// TwinCAT 3 PLC project PLC1
// ProgramVersion: 3.1.4024.0
// libraries:
//   Tc2_Standard, * (Beckhoff Automation GmbH)
//   Tc2_System, * (Beckhoff Automation GmbH)
//   Tc3_Module, * (Beckhoff Automation GmbH)
// project tree:
//   CSL/Enums/ E_Step.TcTLEO
//   CSL/FB/ FB_MSF_Pistons.TcPOU
//   CSL/Structs/ ST_CSL_RawOut.TcDUT, ST_CSL_In.TcDUT, ST_CSL_Out.TcDUT, ST_CSL_Params.TcDUT, ST_CSL_RawIn.TcDUT
//   / PlcTask.TcTTO
//   POUs/ MAIN.TcPOU
// real-time tasks:
//   TASK PlcTask: cycle T#10ms, priority 20, ADS port 350
// motion (NC):
//   TASK NC-Task 1 SAF: cycle T#2ms, priority 4, ADS port 501
//   TASK NC-Task 1 SVB: cycle T#10ms, priority 8, ADS port 511
//   AXIS Asse 1 (id 1)
//     OtherSettings: AllowMotionCmdToSlave=true
//     encoder EncType=4
//       EncPara: MaxCount=#x0000ffff
//         Inc: RefSoftSyncMask=#x0000ffff
//     drive DrvType=24
//       Analog: TorqueSetpointScale=10, ScaleFactorActTorque=0.1
//       TimeComp: TaskDelayCycles=1
//     controller CtrType=1
//       CtrPara: PriorControlFactor=1
//         Observer: BandWidth=20
//   AXIS Asse 2 (id 2)
//     OtherSettings: AllowMotionCmdToSlave=true
//     encoder EncType=4
//       EncPara: MaxCount=#x0000ffff
//         Inc: RefSoftSyncMask=#x0000ffff
//     drive DrvType=24
//       Analog: TorqueSetpointScale=10, ScaleFactorActTorque=0.1
//       TimeComp: TaskDelayCycles=1
//     controller CtrType=1
//       CtrPara: PriorControlFactor=1
//         Observer: BandWidth=20
//   AXIS Asse 3 (id 3)
//     OtherSettings: AllowMotionCmdToSlave=true
//     encoder EncType=4
//       EncPara: MaxCount=#x0000ffff
//         Inc: RefSoftSyncMask=#x0000ffff
//     drive DrvType=24
//       Analog: TorqueSetpointScale=10, ScaleFactorActTorque=0.1
//       TimeComp: TaskDelayCycles=1
//     controller CtrType=1
//       CtrPara: PriorControlFactor=1
//         Observer: BandWidth=20
// I/O:
//   DEVICE Dispositivo 1 (EtherCAT), AmsNetId 5.85.197.242.2.1
//     Terminale 1 (EK1200) [EK1200-5000 EtherCAT Power supply (2A E-Bus)]
//       Terminale 2 (EL1809) [EL1809 16Ch. Dig. Input 24V, 3ms]
//       Terminale 3 (EL2809) [EL2809 16Ch. Dig. Output 24V, 0.5A]
//       Terminale 4 (EL3201) [EL3201 1Ch. Ana. Input PT100 (RTD)]
//       Terminale 5 (EL3311) [EL3311 1Ch. Ana. Input Thermocouple (TC)]
//       Terminale 6 (EL3004) [EL3004 4Ch. Ana. Input +/-10V]
//       Terminale 7 (EL1918) [EL1918, 8Ch. Safety Input 24V, TwinSAFE]
//         modules: Module 1 (FSOE), Module 2 (FSLOGIC)
//       Terminale 8 (EL2904) [EL2904, 4 Ch. Safety Output 24V, 0.5A, TwinSAFE]
//         modules: Module 1 (FSOES), Module 2 (DO)
//       Terminale 9 (EL9011) [EL9011 End Terminal]
//   DEVICE Dispositivo 4 (EtherCAT), AmsNetId 5.85.197.242.5.1
//     Terminale 10 (EK1100) [EK1100 EtherCAT Coupler (2A E-Bus)]
//       Terminale 11 (EL1809) [EL1809 16Ch. Dig. Input 24V, 3ms]
//       Terminale 12 (EL2809) [EL2809 16Ch. Dig. Output 24V, 0.5A]
//       Terminale 13 (EL1809) [EL1809 16Ch. Dig. Input 24V, 3ms]
//       Terminale 14 (EL2809-0015) [EL2809-0015 16Ch. Dig. Output 24V DC, 0.35A, not short-circuit proof]
//       Terminale 15 (EL3202) [EL3202 2Ch. Ana. Input PT100 (RTD)]
//       Terminale 16 (EL3312) [EL3312 2Ch. Ana. Input Thermocouple (TC)]
//       Terminale 17 (EL3632) [EL3632 2Ch. IEPE Sensor]
//       Terminale 18 (EL7031) [EL7031 1Ch. Stepper motor output stage (24V, 1.5A)]
//       Terminale 10 (EL9011) [EL9011 End Terminal]
// variable links:
//   NC-Task 1 SAF/Axes/Asse 3 <-> Device 4 (EtherCAT)/Term 10 (EK1100)/Term 18 (EL7031)
//     Drive/Inputs/In/nState1 @bit 3 <-> STM Status/Status/Error
//     Drive/Inputs/In/nState1 @bit 5 <-> STM Status/Status/Moving negative
//     Drive/Inputs/In/nState1 @bit 4 <-> STM Status/Status/Moving positive
//     Drive/Inputs/In/nState1 @bit 1 <-> STM Status/Status/Ready
//     Drive/Inputs/In/nState1 <-> STM Status/Status/Ready to enable
//     Drive/Inputs/In/nState1 @bit 6 <-> STM Status/Status/Torque reduced
//     Drive/Inputs/In/nState1 @bit 2 <-> STM Status/Status/Warning
//     Drive/Inputs/In/nState2 @bit 3 <-> STM Status/Status/Digital input 1
//     Drive/Inputs/In/nState2 @bit 4 <-> STM Status/Status/Digital input 2
//     Drive/Inputs/In/nState2 @bit 5 <-> STM Status/Status/Sync error
//     Drive/Inputs/In/nState2 @bit 7 <-> STM Status/Status/TxPDO Toggle
//     Drive/Inputs/In/nState4 @bit 1 <-> WcState/InputToggle
//     Drive/Inputs/In/nState4 <-> WcState/WcState
//     Drive/Outputs/Out/nCtrl1 <-> STM Control/Control/Enable
//     Drive/Outputs/Out/nCtrl1 @bit 2 <-> STM Control/Control/Reduce torque
//     Drive/Outputs/Out/nCtrl1 @bit 1 <-> STM Control/Control/Reset
//     Drive/Outputs/Out/nDataOut2[0] <-> STM Velocity/Velocity
//     Enc/Inputs/In/nDataIn1[0] <-> ENC Status compact/Counter value
//     Enc/Inputs/In/nDataIn2[0] <-> ENC Status compact/Latch value
//     Enc/Inputs/In/nState1 @bit 4 <-> ENC Status compact/Status/Counter overflow
//     Enc/Inputs/In/nState1 @bit 3 <-> ENC Status compact/Status/Counter underflow
//     Enc/Inputs/In/nState1 @bit 1 <-> ENC Status compact/Status/Latch extern valid
//     Enc/Inputs/In/nState1 @bit 2 <-> ENC Status compact/Status/Set counter done
//     Enc/Inputs/In/nState2 @bit 4 <-> ENC Status compact/Status/Status of extern latch
//     Enc/Inputs/In/nState2 @bit 5 <-> ENC Status compact/Status/Sync error
//     Enc/Inputs/In/nState2 @bit 7 <-> ENC Status compact/Status/TxPDO Toggle
//     Enc/Inputs/In/nState4 @bit 1 <-> WcState/InputToggle
//     Enc/Inputs/In/nState4 <-> WcState/WcState
//     Enc/Outputs/Out/nCtrl1 @bit 3 <-> ENC Control compact/Control/Enable latch extern on negative edge
//     Enc/Outputs/Out/nCtrl1 @bit 1 <-> ENC Control compact/Control/Enable latch extern on positive edge
//     Enc/Outputs/Out/nCtrl1 @bit 2 <-> ENC Control compact/Control/Set counter
//     Enc/Outputs/Out/nDataOut1[0] <-> ENC Control compact/Set counter value
//   PLC1/PLC1 Instance <-> Device 1 (EtherCAT)/Term 1 (EK1200)/Term 2 (EL1809)
//     PlcTask Inputs/MAIN.stRawIn.bMotorImpulse <-> Channel 1/Input
//     PlcTask Inputs/MAIN.stRawIn.bPieceSensorInput <-> Channel 2/Input
//     PlcTask Inputs/MAIN.stRawIn.bSlot1 <-> Channel 5/Input
//     PlcTask Inputs/MAIN.stRawIn.bSlot2 <-> Channel 6/Input
//     PlcTask Inputs/MAIN.stRawIn.bSlot3 <-> Channel 7/Input
//   PLC1/PLC1 Instance <-> Device 1 (EtherCAT)/Term 1 (EK1200)/Term 3 (EL2809)
//     PlcTask Outputs/MAIN.stRawOut.bCompressor <-> Channel 2/Output
//     PlcTask Outputs/MAIN.stRawOut.bMotor <-> Channel 1/Output
//     PlcTask Outputs/MAIN.stRawOut.bValveSlot1 <-> Channel 3/Output
//     PlcTask Outputs/MAIN.stRawOut.bValveSlot2 <-> Channel 4/Output
//     PlcTask Outputs/MAIN.stRawOut.bValveSlot3 <-> Channel 5/Output

CONFIGURATION PLC1
    RESOURCE PLC ON TwinCAT3
        TASK PlcTask(INTERVAL := T#10ms, PRIORITY := 20);
        PROGRAM MAIN WITH PlcTask : MAIN;
    END_RESOURCE
END_CONFIGURATION

// ---- CSL/Enums/E_Step.TcTLEO
{attribute 'qualified_only'}
{attribute 'strict'}
TYPE E_Step :
(
	(* special steps *)
	NoStep := -32767, // nessuno step    
	Unknown := -32000, // step sconosciuto
	
	(* Not Enabled or Errors*)    
	NeOrError := -990, // non abilitata o in errore
	
	(* Stop *)   
	Stop := 0, // stop
	
	
	conveyor	 :=  130,	//nastro trasportare
	waiting		:= 140,		//attesa
	piston		 := 150		//pistone

);
END_TYPE
//  NoStep = '-32767'
//  Unknown = '-32000'
//  NeOrError = '-990'

// ---- CSL/Structs/ST_CSL_RawOut.TcDUT
TYPE ST_CSL_RawOut :
STRUCT
	(*Digital Outputs*)
	bMotor 			AT %Q*	:	BOOL;	//Q1
	bCompressor 	AT %Q*	:	BOOL;	//Q2
	bValveSlot1 	AT %Q*	:	BOOL;	//Q3
	bValveSlot2 	AT %Q*	:	BOOL;	//Q4
	bValveSlot3		AT %Q*	:	BOOL;	//Q5
	                                         
	bLStart 		AT %Q*	:	BOOL;	//Q9 
	bLStop			AT %Q*	:	BOOL;	//Q10
	bLAck 			AT %Q*	:	BOOL;	//Q11
END_STRUCT
END_TYPE

// ---- CSL/Structs/ST_CSL_In.TcDUT
TYPE ST_CSL_In :
STRUCT
	(*Digital Inputs*)
	bMotorImpulse 		:	BOOL;	//I1  (NC)
	bPieceSensorInput 	:	BOOL;	//I2  (NC)
	bPieceSensorOutput 	:	BOOL;	//I3  (NO)
	bSlot1 				:	BOOL;	//I5  (NC)
	bSlot2 				:	BOOL;	//I6  (NC)
	bSlot3				:	BOOL;	//I7  (NC)
	                    
	bStart 				:	BOOL;	//I9  (NO)
	bStop				:	BOOL;	//I10 (NC)
	bAck 				:	BOOL;	//I11 (NO)
	bEmerg 				:	BOOL;	//12  (NC)
	                    
	(*Analog Input*)    
	nColorSensor		:	REAL;	//I4
	
END_STRUCT
END_TYPE

// ---- CSL/Structs/ST_CSL_Out.TcDUT
TYPE ST_CSL_Out :
STRUCT
	(*Digital Outputs*)
	bMotor 			:	BOOL;	//Q1
	bCompressor 	:	BOOL;	//Q2
	bValveSlot1 	:	BOOL;	//Q3
	bValveSlot2 	:	BOOL;	//Q4
	bValveSlot3		:	BOOL;	//Q5
	                                 
	bLStart 		:	BOOL;	//Q9 
	bLStop			:	BOOL;	//Q10
	bLAck 			:	BOOL;	//Q11
END_STRUCT
END_TYPE

// ---- CSL/Structs/ST_CSL_Params.TcDUT
TYPE ST_CSL_Params :
STRUCT
	StepSlot1			:	INT	:= 	150;
	StepSlot2			:	INT	:= 	160;
	StepSlot3			:	INT	:= 	170;
	StepNoSlot			:	INT	:=	000;
	
	ImpulsePerRotation	:	INT	:=	123;

	
END_STRUCT
END_TYPE

// ---- CSL/Structs/ST_CSL_RawIn.TcDUT
TYPE ST_CSL_RawIn :
STRUCT
	(*Digital Inputs*)
	bMotorImpulse 		AT %I*	:	BOOL;	//I1  (NC)
	bPieceSensorInput 	AT %I*	:	BOOL;	//I2  (NC)
	bPieceSensorOutput 	AT %I*	:	BOOL;	//I3  (NO)
	bSlot1 				AT %I*	:	BOOL;	//I5  (NC)
	bSlot2 				AT %I*	:	BOOL;	//I6  (NC)
	bSlot3				AT %I*	:	BOOL;	//I7  (NC)
	
	bStart 				AT %I*	:	BOOL;	//I9  (NO)
	bStop				AT %I*	:	BOOL;	//I10 (NC)
	bAck 				AT %I*	:	BOOL;	//I11 (NO)
	bEmerg 				AT %I*	:	BOOL;	//12  (NC)
	
	(*Analog Input*)
	nColorSensor		AT %I*	:	INT;	//I4
END_STRUCT
END_TYPE

// ---- POUs/MAIN.TcPOU
PROGRAM MAIN


VAR
	stRawIn		:	ST_CSL_RawIn;
	stRawOut	:	ST_CSL_RawOut;
	stIn		:	ST_CSL_In;
	stOut		: 	ST_CSL_Out;
	stParams	:	ST_CSL_Params; 
	fbPistons	: FB_MSF_Pistons;
	
	estep 	: E_Step;
	
	
	slots	: INT;
	nerrid	: DINT; 
	bfbend : BOOL;
	
END_VAR

stIn.bMotorImpulse 			:= stRawIn.bMotorImpulse 		;
stIn.bPieceSensorInput 		:= stRawIn.bPieceSensorInput 	;
stIn.bPieceSensorOutput 	:= stRawIn.bPieceSensorOutput 	;	
stIn.bSlot1 				:= stRawIn.bSlot1 				;	
stIn.bSlot2 				:= stRawIn.bSlot2 				;	
stIn.bSlot3	            	:= stRawIn.bSlot3				; 
stIn.bStart 				:= stRawIn.bStart               ;    	
stIn.bStop					:= stRawIn.bStop	 			;	
stIn.bAck 					:= stRawIn.bAck 				;
stIn.bEmerg 				:= stRawIn.bEmerg				;
                                        				

fbPistons(
	bEnable		:=  TRUE, 
	slot 		:= slots, 
	st_In 		:= stIn, 
	st_Params 	:= stParams, 
	eStep		=> estep, 
	eErrStep	=> estep, 
	nErrid		=> nerrid, 
	bFbEnd		=> bfbend);
	

stRawOut :=  fbPistons.st_Out;

END_PROGRAM

// ---- CSL/FB/FB_MSF_Pistons.TcPOU
FUNCTION_BLOCK FB_MSF_Pistons
VAR_INPUT
	bEnable	: BOOL;
	slot	: INT;

END_VAR

VAR_IN_OUT
	
	st_In		:	ST_CSL_In;
	st_Params	: 	ST_CSL_Params;
	
	
END_VAR


VAR_OUTPUT
	
	eStep	: E_Step;		//current step of the state machine
	eErrStep : E_Step;  //step where an error was raised
	nErrid	: DINT;		//error identification code
	
	bFbEnd	:	BOOL;
	
	st_Out		: 	ST_CSL_RawOut;
	
	END_VAR
VAR
	bSensor: BOOL;
	bValve : BOOL;
	nStepSlot : INT;
	Timer_Pistons : TON();
	Error: DINT;
	iMotor	: INT := 0;
    

	bInitialized	: BOOL;		//FB initialization
	eNewStep : E_Step;			//request for a new step
	bEntryact	: 	BOOL;		//step entry action performed
	
	fbRtMotorImpulse	: R_TRIG;
	
		
	
END_VAR

(* initialization *)
IF NOT bInitialized THEN    
	eNewstep 		:= 	E_Step.NoStep;    
	eStep 			:= 	E_Step.Conveyor;    
	bEntryact 		:= 	FALSE;    
	bInitialized 	:= 	TRUE; 
	bFbEnd			:=	FALSE;

	// association of the motors and the sensors to the steps
	CASE slot OF
		0:
			nStepSlot	:=	st_Params.StepNoSlot;	
		1:
			bValve		:= 	st_Out.bValveSlot1;
			bSensor 	:= 	st_In.bSlot1;
			nStepSlot 	:= 	st_Params.StepSlot1;
		2:
			bValve		:= 	st_Out.bValveSlot2;
			bSensor 	:= 	st_In.bSlot2;
			nStepSlot 	:= 	st_Params.StepSlot2;
		3:
			bValve		:= 	st_Out.bValveSlot3;
			bSensor 	:= 	st_In.bSlot3;
			nStepSlot 	:= 	st_Params.StepSlot3;
			
	END_CASE


ELSE   

	(* forcing the error state *)	
	(* disabled or faulty *)
	IF  NOT bEnable THEN
		eNewstep 	:=	E_Step.NeOrError;

	END_IF;

	(* state change managementstate change management *)
	IF eNewstep <> E_Step.NoStep THEN    
		eStep 		:= 	eNewstep;    
		eNewstep 	:= 	E_Step.NoStep;   
 		bEntryact 	:= 	FALSE;

	END_IF;

	
	(* input signal conditioning *)
	(*filters*)
	Timer_Pistons (IN:= (iMotor = nStepSlot), PT := T#500MS);
	(*fronts*)
	//fbRtMotorImpulse(CLK:=	st_In.bMotorImpulse );

	// storing of the pieces
	CASE eStep OF

		// conveyor of the pieces
		E_Step.conveyor :
	
			(* body *)	
			st_Out.bMotor		:=	 TRUE;
			st_Out.bCompressor 	:=	 TRUE;
			bValve 				:=	 FALSE;	
			
			(*Counter of steps*)
			IF st_In.bMotorImpulse	THEN
				iMotor := iMotor + 1;
			END_IF
		
			(* transition *)	
			IF bEnable THEN          
		 		eNewstep := E_Step.NeOrError;        
			ELSE 
				IF  iMotor = nStepSlot THEN 
					eNewstep := E_Step.waiting;            
        		END_IF;
			END_IF
	
		// waiting of the movement of the piston
		E_Step.waiting :
	
			(* body *)
			st_Out.bMotor		:=	FALSE;
			st_Out.bCompressor 	:= 	TRUE;
			bValve 				:=	FALSE;	
			iMotor := 0;
		
			(* transition *)
			IF bEnable THEN          
		 		eNewstep := E_Step.NeOrError;        
			ELSE 
				IF  Timer_Pistons.Q THEN 
					eNewstep := E_Step.piston;            
       	 		END_IF;
			END_IF	
	
		// activation of the motors of the pistons.
		E_Step.piston :

			(* body *)
			st_Out.bMotor		:= 	FALSE;
			st_Out.bCompressor 	:= 	TRUE;
			bValve 				:=	TRUE;
	
			(* transition *)
			IF bEnable THEN          
		 		eNewstep := E_Step.NeOrError;        
			ELSE 
				IF  NOT bsensor THEN 
					bFbEnd	:= TRUE;         
       	 			END_IF;
			END_IF
	
	
		ELSE
	
		// Error case
		eNewstep 	:= 	E_Step.NeOrError;
		eErrStep 	:=	E_Step.Unknown;
		nErrId 		:= 	-9; 	
		
		
	END_CASE


END_IF

END_FUNCTION_BLOCK
